{attribute 'GeneratedUsingTerminal: AT2050-0500-0018'}
{attribute addProperty BoxType "AT2050-0500-0018"}
{attribute addProperty Id "A_0095_AT2021_5250_0019_AT2021_5250AT2021_01D6DEDF80"}
{attribute addProperty CRC "1501147460"}
{attribute addProperty Size "80"}
TYPE A_0049_AT2050_0500_0018_5979B144 EXTENDS AT2050_86175B41 :
STRUCT
	{attribute addProperty Name "A_0095_AT2021_5250_0019_AT2021_5250"}
	{attribute addProperty PreviousPort "A_0049(AT2050-0500-0018) : B"}
	A_0095_AT2021_5250_0019_AT2021_5250 : AT2021_01D6DEDF;
END_STRUCT
END_TYPE

(* stored: Version 1.2.0.0, ProductVersion 3.1.4024.9
   DUT A_0049_AT2050_0500_0018_5979B144: Id {f86404eb-0169-47b7-a4f4-5cc6bd24f475} *)
